{attribute 'qualified_only'}
VAR_GLOBAL
	bSendDoneFiFo	:ARRAY[1..cMaxRS485CMDFiFo] OF BOOL;			(* Rückmeldung Aus dem FiFo Master Baustein, dass der Sendevorgang abgeschlossen ist *)
	sSendFiFo		:ARRAY[1..cMaxRS485CMDFiFo] OF STRING(255);		(* Zeile für den FiFo Master Baustein, von jedem einzelnen Busteilnehmer *)
END_VAR

(* stored: Version 1.1.0.1, ProductVersion 3.1.4024.12
   GVL GVL_RS485FiFoSend: Id {8564bc8f-e893-47d7-8bf8-1cb12d584f70} *)
